// TIA Portal V16 export
// export: Created 2021-07-12T14:47:19.5871213Z, ExportSetting WithDefaults, DisplayName Totally Integrated Automation Portal, DisplayVersion V16, DisplayName TIA Portal Version Control Interface, DisplayVersion V16, DisplayName TIA Portal Openness, DisplayVersion V16, DisplayName STEP 7 Professional, DisplayVersion V16, DisplayName STEP 7 Safety, DisplayVersion V16, DisplayName WinCC Professional, DisplayVersion V16
TYPE "LSimaHydTO_typeForceLimits"
TITLE = LSimaHydTO_typeForceLimits
// Force limits
// stored: IsFailsafeCompliant false
   STRUCT
      MaxForce { S7_SetPoint := 'True'} : LReal := 100.0;   // Maximum force
      MaxForceRamp { S7_SetPoint := 'True'} : LReal := 10000.0;   // Force increase limitation
   END_STRUCT;
END_TYPE
